PROGRAM MAIN
VAR

cbBlock1 : CommandBlockBase;
cbBlock2 : CommandBlockBase;

cbBlock3 : CommandBlockPos;
cbBlock4 : CommandBlockPos;

ptBlock : POINTER TO CommandBlockBase := ADR(cbBlock1);	
ptBlockPos : POINTER TO CommandBlockPos;

aSize : INT;


memoryPool : ARRAY[1..1024] OF WORD;

ptRunIndexerMaster : POINTER TO RunUnitIndexerMaster;
ptRunGeneric : POINTER TO RunUnitGeneric;

ptUnitGeneric : POINTER TO UnitBase;
ptUnitIndexerMaster : POINTER TO UnitIndexerMaster;


END_VAR

cbBlock1.AXIS_ID:=5;
MAIN.ptBlock:=ADR(cbBlock1);

cbBlock2:=MAIN.ptBlock^; // value assignment?
//change cbBlock1 , watch if cbBlock2 changed

MAIN.ptBlock := ADR(cbBlock3); //if possible mophism

cbBlock3.COORDINATE:=1234;

ptBlockPos:=MAIN.ptBlock;
cbBlock4:=ptBlockPos^;//check


//may access violation??
//ptBlockPos:=ADR(cbBlock1);
//ptBlockPos^.COORDINATE:=5555; //may violation

//TEST2();
//TEST_CYLINDER();
//TEST_UNIT_VIRTUAL();
//TEST_UNIT_MASTER();

aSize := SIZEOF(GVL.unitControls[1]);
aSize := SIZEOF(UnitBase);
aSize := SIZEOF(UnitIndexerMaster);
//fbCylinder(ptBlock:= ADR(cylinderBlock));

//fbRunIndexerMaster(ptBlock:= );


//no need
//ptRunIndexerMaster := ADR(memoryPool[1]); // fine?
//ptRunGeneric := ADR(memoryPool[1+SIZEOF(ptRunIndexerMaster)]);

//ptRunIndexerMaster^();
//ptRunGeneric^();


//possible manipulate memory allocation
ptUnitGeneric := ADR(memoryPool[1]);
ptUnitIndexerMaster := ADR(memoryPool[1+SIZEOF(ptUnitGeneric^)]);

ptUnitGeneric^.alarmCode := 99;  //

METHOD FB_init : BOOL
VAR_INPUT
	bInitRetains : BOOL; // if TRUE, the retain variables are initialized (warm start / cold start)
	bInCopyCode : BOOL;  // if TRUE, the instance afterwards gets moved into the copy code (online change)
END_VAR
END_METHOD

END_PROGRAM

(* stored: Version 1.1.0.1, ProductVersion 3.1.4020.12
   POU MAIN: Id {c5d24ec2-dcd4-432d-b366-2840b187b342}, SpecialFunc None
   Method FB_init: Id {9aee4cb1-a42d-4360-bcd2-e6043699c579} *)
